// TIA Portal V21 export
FUNCTION "GestAdditivo" : Void   // FC84, LAD
{ S7_Optimized_Access := 'TRUE' }
// stored: SetENOAutomatically false
   VAR_INPUT
      "K_Analogica(Mandata)" : Int;   // K_Analogica della pompa di mandata prodotto
      K_Pid : Int;
      "K_Motore(Additivo)" : Int;   // K_Motore della pompa dell'additivo
      K_Additivo : Int;   // K_Additivo attuale
   END_VAR
   VAR_TEMP
      AppoggioPortata : Real;
      AppoggioCalcoli : Real;
      PortataAdditivoNecessaria : Real;
      HzPompaAdditivoNecessari : Real;
      "PortataAttualeTeorica(l/h)" : Real;
      "PortataAttualeTeorica(ql.i/h)" : Real;
      AdditivoAllaMassimaVel : Bool;
      VelRichiesta : Real;
      VelAttualeHzFromScale : Real;
      K_AnalogicaInt : Int;
      K_MotoreInt : Int;
      K_AdditivoInt : Int;
      K_PidInt : Int;
   END_VAR
   VAR CONSTANT
      FrequenzaMinInv : Real := 10.0;
      FrequenzaMaxInv : Real := 80.0;
      MassimaPortataPompa : Real := 271.0;
      MinimaPortataPompa : Real := 30.0;
   END_VAR
BEGIN

REGION Network 1 (SCL): Calcolo e scalatura percentuale acido
   REGION Diagnostica programmatore
       (*Passiamo tutte le costanti di accesso agli array in modo da verificarle e controllarle*)
       "Diagnostica"(K_Attuale_ArrayInCuiAccediamo :=  #"K_Analogica(Mandata)",
                     K_NumMax_MassimoValoreDellArrayInCuiAccediamo := "K_NumAnalogica",
                     K_Tipo_ArrayInCuiAccediamo := "K_TipoAnalogica",
                     K_Attuale_DiChiAccede := #"K_Analogica(Mandata)",
                     K_Tipo_DiChiAccede := "K_TipoAdditivo",
                     K_AttualeInterno => #K_AnalogicaInt);

       "Diagnostica"(K_Attuale_ArrayInCuiAccediamo := #"K_Motore(Additivo)",
                     K_NumMax_MassimoValoreDellArrayInCuiAccediamo := "K_NumMotore",
                     K_Tipo_ArrayInCuiAccediamo := "K_TipoMotore",
                     K_Attuale_DiChiAccede := #"K_Motore(Additivo)",
                     K_Tipo_DiChiAccede := "K_TipoAdditivo",
                     K_AttualeInterno => #K_MotoreInt);

       "Diagnostica"(K_Attuale_ArrayInCuiAccediamo := #K_Additivo,
                     K_NumMax_MassimoValoreDellArrayInCuiAccediamo := "K_NumAdditivo",
                     K_Tipo_ArrayInCuiAccediamo := "K_TipoAdditivo",
                     K_Attuale_DiChiAccede := #K_Additivo,
                     K_Tipo_DiChiAccede := "K_TipoAdditivo",
                     K_AttualeInterno => #K_AdditivoInt);

       "Diagnostica"(K_Attuale_ArrayInCuiAccediamo := #K_Pid,
                     K_NumMax_MassimoValoreDellArrayInCuiAccediamo := "K_NumPid",
                     K_Tipo_ArrayInCuiAccediamo := "K_TipoPid",
                     K_Attuale_DiChiAccede := #K_Pid,
                     K_Tipo_DiChiAccede := "K_TipoAdditivo",
                     K_AttualeInterno => #K_PidInt);
   END_REGION ;
   REGION Calcolo portata acido necessario in quintali/h
       #"PortataAttualeTeorica(l/h)":=
       #PortataAdditivoNecessaria := "Analogica".A[#K_AnalogicaInt].Out.AnalogicaAttuale.Valore / 100.0 * "Additivo".A[#K_AdditivoInt].Prm.PercentualeAdditivoRich;
   END_REGION ;
   REGION Calcolo e parametrizzo valori PID
       "Pid".P[#K_Pid].Hmi.SetpointFF := #PortataAdditivoNecessaria;
       "Pid".P[#K_Pid].Prm.FF.interpolazione[0].Setpoint := #MinimaPortataPompa;
       "Pid".P[#K_Pid].Prm.FF.interpolazione[0].Valore := #FrequenzaMinInv;
       "Pid".P[#K_Pid].Prm.FF.interpolazione[1].Setpoint := #MassimaPortataPompa;
       "Pid".P[#K_Pid].Prm.FF.interpolazione[1].Valore := #FrequenzaMaxInv;
   END_REGION ;
   REGION Allarmi
       IF #PortataAdditivoNecessaria > #MassimaPortataPompa THEN
           "Additivo".A[#K_AdditivoInt].Allarmi.A[KALLAdditivo_PortataPrincipaleTroppoAlta].Stato := True;
           #"PortataAttualeTeorica(l/h)" := #MassimaPortataPompa;
       END_IF;
       IF #PortataAdditivoNecessaria < #MinimaPortataPompa THEN
           "Additivo".A[#K_AdditivoInt].Allarmi.A[KALLAdditivo_PortataPrincipaleTroppoBassa].Stato := True;
           #"PortataAttualeTeorica(l/h)" := #MinimaPortataPompa;
       END_IF;
   END_REGION ;
   REGION Calcolo portata additivo attuale     
       #"PortataAttualeTeorica(ql.i/h)" := #"PortataAttualeTeorica(l/h)" / 100.0;
       "Additivo".A[#K_AdditivoInt].Out.AttualeAdditivo := #"PortataAttualeTeorica(ql.i/h)";
       IF NOT "Motore".M[#"K_Motore(Additivo)"].Out.InMarcia THEN
           "Additivo".A[#K_AdditivoInt].Out.AttualeAdditivo := 0.0;
       END_IF;
   END_REGION ;
END_REGION
END_FUNCTION
